TYPE SharedContextCom :
STRUCT
  Publish : SharedContextComPublish;
  Subscribe : SharedContextComSubscribe;
END_STRUCT
END_TYPE

(* stored: Version 1.1.0.1
   DUT SharedContextCom: Id {3482cefa-34e6-4ed4-ad10-8cc96dfa7a43} *)
